Omron Sysmac Studio project ExampleUDPSocket (Sysmac Studio 1.63.0.7, StandardProject)

# Controller Example: NX102-9000 version 1.64
Task PrimaryTask (priority 4, period or condition 2000): Main

PROGRAM Main
VAR
    iSktUDPCreaate : SktUDPCreate;
    iSktUDPSend : SktUDPSend;
    iSktClose : SktClose;
END_VAR
VAR CONSTANT
    STATE_ERROR : UINT := 900;
    STATE_CLOSE : UINT := 990;
    STATE_DONE : UINT := 1000;
END_VAR
VAR
    DESTINATIONS : ARRAY[0..3] OF _sSOCKET_ADDRESS;
    iState : UINT;
    iSocket : _sSOCKET;
    iData : ARRAY[0..1023] OF BYTE;
    iDataSize : UINT;
    iCounter : UDINT;
    iDestSelection : UINT;
    iErrorState : UINT;
    iError : BOOL;
    iErrorID : WORD;
    iWaitTick : UINT;
END_VAR
CASE iState OF
	// STATE_INIT
	0:
		// 送信先設定
		DESTINATIONS[0].IpAdr := '192.168.250.*'; DESTINATIONS[0].PortNo := 15001;
		DESTINATIONS[1].IpAdr := '192.168.250.*'; DESTINATIONS[1].PortNo := 15002;
		DESTINATIONS[2].IpAdr := '192.168.250.*'; DESTINATIONS[2].PortNo := 15003;
		DESTINATIONS[3].IpAdr := '192.168.250.*'; DESTINATIONS[3].PortNo := 15004;

		// FBを初期化
		iSktUDPCreaate.Execute := FALSE;
		iSktUDPSend.Execute := FALSE;
		iSktClose.Execute := FALSE;
		
		Clear(iSocket);
		Clear(iCounter);
		Clear(iData);
		Clear(iDataSize);
		Clear(iDestSelection);
		Clear(iError);
		Clear(iErrorID);
		Clear(iWaitTick);
		
		Inc(iState);
	1:
		iSktUDPCreaate.SrcUdpPort := 15001;
		iSktUDPCreaate.Execute := TRUE;
		
		Inc(iState);
	2:
		IF iSktUDPCreaate.Done OR iSktUDPCreaate.Error THEN
			iSktUDPCreaate.Execute := FALSE;
			
			IF iSktUDPCreaate.Error THEN
				iErrorState := iState;
				iError := TRUE;
				iErrorID := iSktUDPCreaate.ErrorID;
				iState := STATE_ERROR;
			ELSE
				// 生成したSocketを保存
				iSocket := iSktUDPCreaate.Socket;
				
				Inc(iState);
			END_IF;
		END_IF;
	3:
		// 送信先を都度変更
		iSocket.DstAdr := DESTINATIONS[iDestSelection];
		iDestSelection := (iDestSelection + 1) MOD 4;
		
		Inc(iState);
	4:
		// データ生成
		Inc(iCounter);
		iDataSize := StringToAry(In:=CONCAT(UDINT_TO_STRING(iCounter), '$n'),
								 AryOut:=iData[0]);
		iSktUDPSend.Size := iDataSize;
		
		// 送信処理開始時にSocketを設定
		iSktUDPSend.Socket := iSocket;
		iSktUDPSend.Execute := TRUE;
				
		Inc(iState);
	5:
		IF iSktUDPSend.Done OR iSktUDPSend.Error THEN
			// ソケット命令は、使用後に必ず1サイクルの休止を入れる。
			// 無休止で使用すると数時間～数日の連続稼働後にネットワーク機能全般が機能不全に陥る。
			iSktUDPSend.Execute := FALSE;
			
			IF iSktUDPSend.Error THEN
				iErrorState := iState;
				iError := TRUE;
				iErrorID := iSktUDPSend.ErrorID;
				iState := STATE_ERROR;
			ELSE
				iWaitTick := 500;
				
				Inc(iState);
			END_IF;
		END_IF;
	6:
		Dec(iWaitTick);
		IF iWaitTick < 1 THEN
			iState := iState - 3;
		END_IF;
		
	// STATE_ERROR
	// iErrorState=2: iSktUDPCreateでエラー
	// iErrorState=5: iSktUDPSendでエラー
	900:
		// 何らかのエラー処理
		
		iState := STATE_CLOSE;

	// STATE_CLOSE
	990:
		// Socketは、エラーを生じたものであっても念のため閉じる。
		
		iSktClose.Socket := iSocket;
		iSktClose.Execute := TRUE;
		
		Inc(iState);
	991:
		IF iSktClose.Done OR iSktClose.Error THEN
			iSktClose.Execute := FALSE;
			
			// ソケット通信リソースオーバーで失敗した場合、再実行する。
			// リソースオーバーは、ソケット命令同時実行数を超過しているだけ。
			IF iSktClose.Error AND iSktClose.ErrorID = WORD#16#2008 THEN
				Dec(iState);
			ELSE
				iState := STATE_DONE;
			END_IF;
		END_IF;
	
	// STATE_DONE
	// 1000:
END_CASE;

iSktUDPCreaate();
iSktUDPSend(SendDat:=iData[0]);
iSktClose();
END_PROGRAM